Staubli VAL3: createFrame.pgx

public program createFrame(frame x_fFrame, bool& x_bError[])
  local num l_nSizeTab
begin
  //Header begin
  //Description of program
  //  This program creates an area for monitoring the Z position of
  //  a tool center point in regards to a frame.
  //
  //Input parameters
  //  frame x_fFrame :
  //    role : defines the frame that you want to use for monitoring the z value
  //
  //Output parameters
  //  bool x bError :
  //    role : set to true when the frame area could not be created, false otherwise
  //
  //Example
  //  call createFrame(fTable,bOK)
  //
  //History
  //  Creation : 16-04-08 - f.Rob
  //Header end


  l_nSizeTab=size(fFrameZone)

  //Test if it's possible to creates a new cylinder (not exceed the maximum size of the array)
  if (nNumberFrame>l_nSizeTab-1)
    x_bError=true
    popUpMsg("Frame area number "+toString("",nNumberFrame)+" cannot be created : you can create only "+toString("",l_nSizeTab)+" (0.."+toString("",l_nSizeTab-1)+") area of this type")
    return
  endIf
  //Build the frame
  fFrameZone[nNumberFrame]=x_fFrame
  bCreateFrame[nNumberFrame]=true

  nNumberFrame=nNumberFrame+1
end
